{attribute addProperty BoxType "EK1100-0000-0018"}
{attribute addProperty Id "Beckhoff_EPP7xxxEK1122Beckhoff_EPP7xxxEK1122_95AA5F572464308"}
{attribute addProperty CRC "2202949598"}
{attribute addProperty SizeInBites "2464"}
{attribute addProperty SizeInBytes "308"}
TYPE Beckhoff_EPP7xxx_834E57DE EXTENDS EK1100_179A0949 :
STRUCT
	{attribute addProperty Name "Beckhoff_EPP7xxxEK1122"}
	Beckhoff_EPP7xxxEK1122 : Beckhoff_EPP7xxxEK1122_95AA5F57;
END_STRUCT
END_TYPE

(* stored: Version 1.2.0.0, ProductVersion 3.1.4024.9
   DUT Beckhoff_EPP7xxx_834E57DE: Id {4857a66a-9d2e-4205-8eea-b2dd7379dcb2} *)
